INTERFACE ITF_Regelschuif_In_DG

METHOD get : SINT
VAR_INPUT
END_VAR
END_METHOD

END_INTERFACE

(* stored: Version 1.1.0.1, ProductVersion 3.1.4026.8
   Itf ITF_Regelschuif_In_DG: Id {9b33a0ca-525b-478a-ac94-1f494bb5dbb6}
   Method get: Id {505b80cc-8804-424e-afea-4cfa6331bd6f} *)
